FUNCTION "LnkJ_Fixture" : Void
{ S7_Optimized_Access := 'TRUE' }
VERSION : 0.1
   VAR_INPUT
      Seq : UInt;   // 엔벨로프 seq (1..65535, 0 = 없음)
   END_VAR

   VAR_IN_OUT
      Buf : Array[*] of Byte;   // 출력 버퍼
      Pos : DInt;   // 다음 쓸 절대 인덱스 (< 0 = 오류 유지)
      Val : "LNK_Fixture";   // data
   END_VAR


BEGIN
	// GENERATED by gr-contract gen-link from message "Fixture" (id 40, "LNK_Fixture" sig 16#EB2E5DE0) - do not edit
	// {"type":"Fixture","seq":<Seq>,"sig":3945684448,"data":<Val>}
	"Json_WRaw"(Buf := #Buf, Pos := #Pos, Lit := '{"type":"Fixture","seq":');
	"Json_WUInt"(Buf := #Buf, Pos := #Pos, Val := #Seq);
	"Json_WRaw"(Buf := #Buf, Pos := #Pos, Lit := ',"sig":3945684448,"data":');
	"JsonW_LNK_Fixture"(Buf := #Buf, Pos := #Pos, Val := #Val);
	"Json_WRaw"(Buf := #Buf, Pos := #Pos, Lit := '}');
END_FUNCTION
